// TIA Portal V17 export
// export: Created 2025-04-11T04:54:25.0955287Z, ExportSetting WithDefaults, DisplayName Totally Integrated Automation Portal, DisplayVersion V17, DisplayName TIA Portal Openness, DisplayVersion V17, DisplayName TIA Portal Version Control Interface, DisplayVersion V17, DisplayName SINAMICS Startdrive Advanced, DisplayVersion V17, DisplayName SINAMICS Startdrive G130, G150, S120, S150, SINAMICS MV, S210, DisplayVersion V17, DisplayName SINAMICS Startdrive G110M, G120, G120C, G120D, G120P, G115D, DisplayVersion V17, DisplayName STEP 7 Professional, DisplayVersion V17, DisplayName STEP 7 Safety, DisplayVersion V17, DisplayName WinCC Advanced, DisplayVersion V17
TYPE "UDT_Ana_PreAlarm"
// stored: IsFailsafeCompliant false
   STRUCT
      OUT_HPreAlarm : Bool;   // 高预警
      OUT_LPreAlarm : Bool;   // 低预警
      OUT_wPreAlarm : Word;   // 预警字 (Bit0=高预警, Bit1=低预警)
   END_STRUCT;
END_TYPE
